FUNCTION_BLOCK FB_Motor
VAR_INPUT
END_VAR
VAR_OUTPUT
END_VAR
VAR
	Value 		: LREAL;
	Parameters 	: ST_MotorParam := (Set := 1, P := 2, I := 3, D := 4, Unit:='%');
END_VAR

Value := HMI.SineVerySlow*100/2;

END_FUNCTION_BLOCK

(* stored: Version 1.1.0.1, ProductVersion 3.1.4022.18
   POU FB_Motor: Id {fe771ada-2e33-42ec-85fa-eac4a5319fc1}, SpecialFunc None *)
